(* IEC 61131-3 sources: POMIRTS_lab3/AS/Library_2/AsSLIP, 3 files *)

(* ---- AsSLIP.typ ---- *)
TYPE
    slipPARAMETER_typ	: STRUCT		(*slip parameter*)
		pHostAddr		: UDINT;		(*pointer to the host ip address (string format)*)
		pPeerAddr		: UDINT;		(*pointer to the peer ip address (string format)*)
		mtu				: UDINT;		(*maximum trasmission unit*)
		compAllow		: BOOL;			(*compression allow*)
		compEnable		: BOOL;			(*compression enable*)
	END_STRUCT;
END_TYPE

(* ---- AsSLIP.fun ---- *)
{REDUND_CONTEXT} {REDUND_UNREPLICABLE} FUNCTION_BLOCK SLIPStart				(*starts a SLIP device; asynchronous execution*)
	VAR_INPUT
		enable			: BOOL;			(*enables execution*)
		pDevice			: UDINT;		(*device name given as a pointer*)
		pDeviceParam	: UDINT;		(*pointer to the parent device parameter (optional)*)
		pSlipParam		: UDINT;		(*pointer to the slip parameter (optional)*)
	END_VAR

	VAR
        i_state			: UINT;			(*internal variable*)
		i_result		: UINT;			(*internal variable*)
        i_tmp			: UDINT;		(*internal variable*)
	END_VAR

	VAR_OUTPUT
		status			: UINT;			(*execution status: ERR_OK, ERR_FUB_ENABLE_FALSE, ERR_FUB_BUSY, 0xXXXX = see help*)
	END_VAR
END_FUNCTION_BLOCK

{REDUND_CONTEXT} {REDUND_UNREPLICABLE} FUNCTION_BLOCK SLIPStop					(*stops a SLIP device; asynchronous execution*)
	VAR_INPUT
		enable			: BOOL;			(*enables execution*)
		pDevice			: UDINT;		(*device name given as a pointer*)
	END_VAR

	VAR
        i_state			: UINT;			(*internal variable*)
		i_result		: UINT;			(*internal variable*)
        i_tmp			: UDINT;		(*internal variable*)
	END_VAR

	VAR_OUTPUT
		status			: UINT;			(*execution status: ERR_OK, ERR_FUB_ENABLE_FALSE, ERR_FUB_BUSY, 0xXXXX = see help*)
	END_VAR
END_FUNCTION_BLOCK

(* ---- AsSLIP.var ---- *)
VAR CONSTANT
	slipERR_INVALID_DEVICE				: UINT := 31950;	(*invlalid parent device*)
END_VAR
